// Mitsubishi GX Works2 project: msp_4   PLC: Q03UDV

PROGRAM MAIN
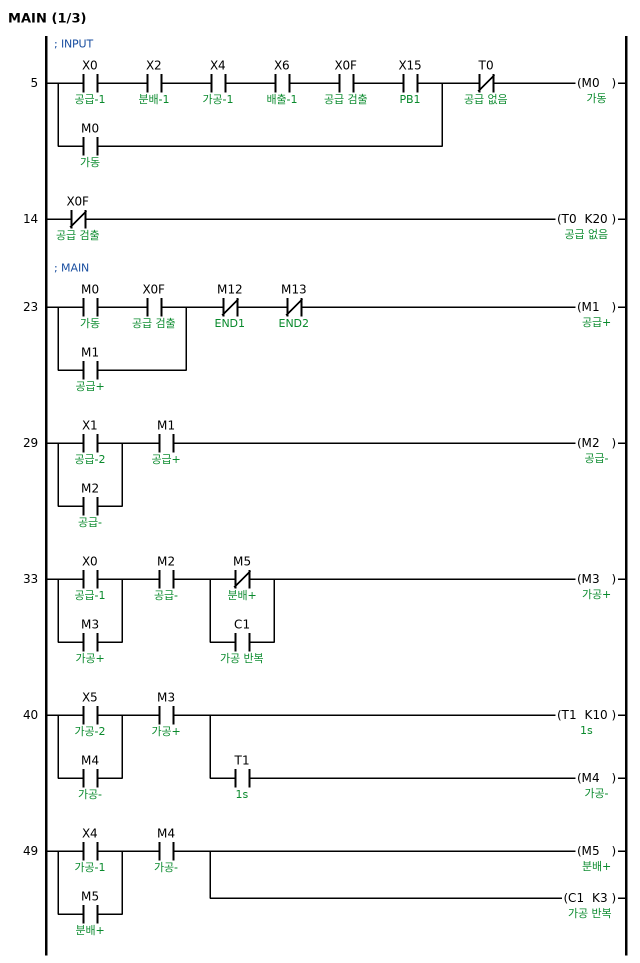
; INPUT
5     LD      X0  ; 공급-1
      AND     X2  ; 분배-1
      AND     X4  ; 가공-1
      AND     X6  ; 배출-1
      AND     X0F  ; 공급 검출
      AND     X15  ; PB1
      OR      M0  ; 가동
      ANI     T0  ; 공급 없음
      OUT     M0  ; 가동
14    LDI     X0F  ; 공급 검출
      OUT     T0 K20  ; 공급 없음
; MAIN
23    LD      M0  ; 가동
      AND     X0F  ; 공급 검출
      OR      M1  ; 공급+
      ANI     M12  ; END1
      ANI     M13  ; END2
      OUT     M1  ; 공급+
29    LD      X1  ; 공급-2
      OR      M2  ; 공급-
      AND     M1  ; 공급+
      OUT     M2  ; 공급-
33    LD      X0  ; 공급-1
      OR      M3  ; 가공+
      AND     M2  ; 공급-
      LDI     M5  ; 분배+
      OR      C1  ; 가공 반복
      ANB
      OUT     M3  ; 가공+
40    LD      X5  ; 가공-2
      OR      M4  ; 가공-
      AND     M3  ; 가공+
      OUT     T1 K10  ; 1s
      AND     T1  ; 1s
      OUT     M4  ; 가공-
49    LD      X4  ; 가공-1
      OR      M5  ; 분배+
      AND     M4  ; 가공-
      OUT     M5  ; 분배+
      OUT     C1 K3  ; 가공 반복
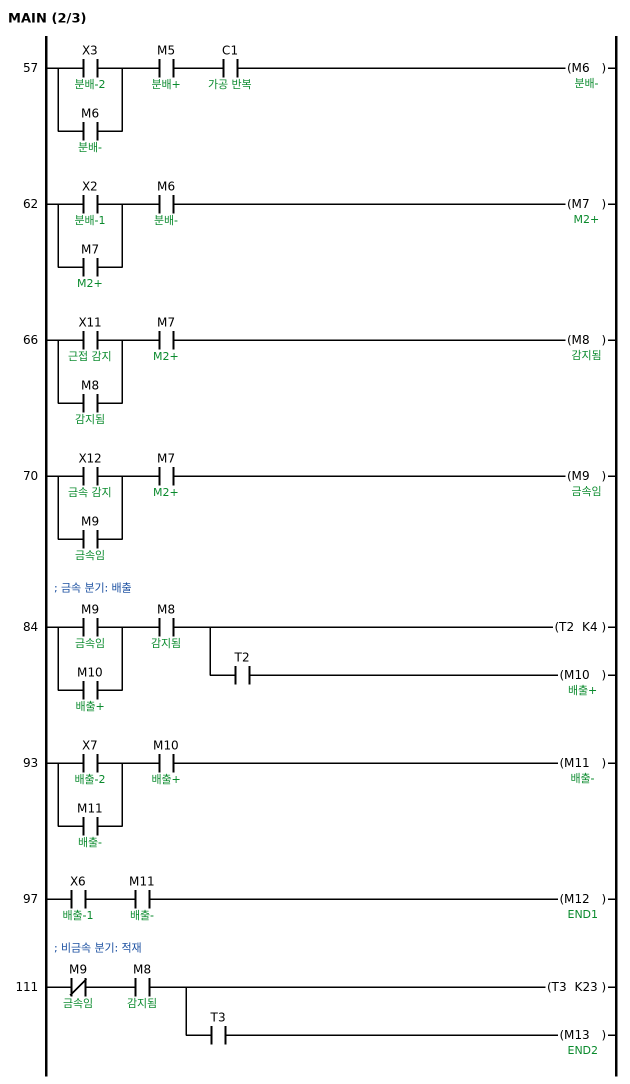
57    LD      X3  ; 분배-2
      OR      M6  ; 분배-
      AND     M5  ; 분배+
      AND     C1  ; 가공 반복
      OUT     M6  ; 분배-
62    LD      X2  ; 분배-1
      OR      M7  ; M2+
      AND     M6  ; 분배-
      OUT     M7  ; M2+
66    LD      X11  ; 근접 감지
      OR      M8  ; 감지됨
      AND     M7  ; M2+
      OUT     M8  ; 감지됨
70    LD      X12  ; 금속 감지
      OR      M9  ; 금속임
      AND     M7  ; M2+
      OUT     M9  ; 금속임
; 금속 분기: 배출
84    LD      M9  ; 금속임
      OR      M10  ; 배출+
      AND     M8  ; 감지됨
      OUT     T2 K4
      AND     T2
      OUT     M10  ; 배출+
93    LD      X7  ; 배출-2
      OR      M11  ; 배출-
      AND     M10  ; 배출+
      OUT     M11  ; 배출-
97    LD      X6  ; 배출-1
      AND     M11  ; 배출-
      OUT     M12  ; END1
; 비금속 분기: 적재
111   LDI     M9  ; 금속임
      AND     M8  ; 감지됨
      OUT     T3 K23
      AND     T3
      OUT     M13  ; END2
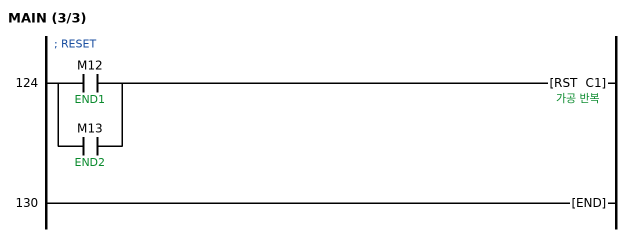
; RESET
124   LD      M12  ; END1
      OR      M13  ; END2
      RST     C1  ; 가공 반복
130   END
END_PROGRAM

PROGRAM OUTPUT
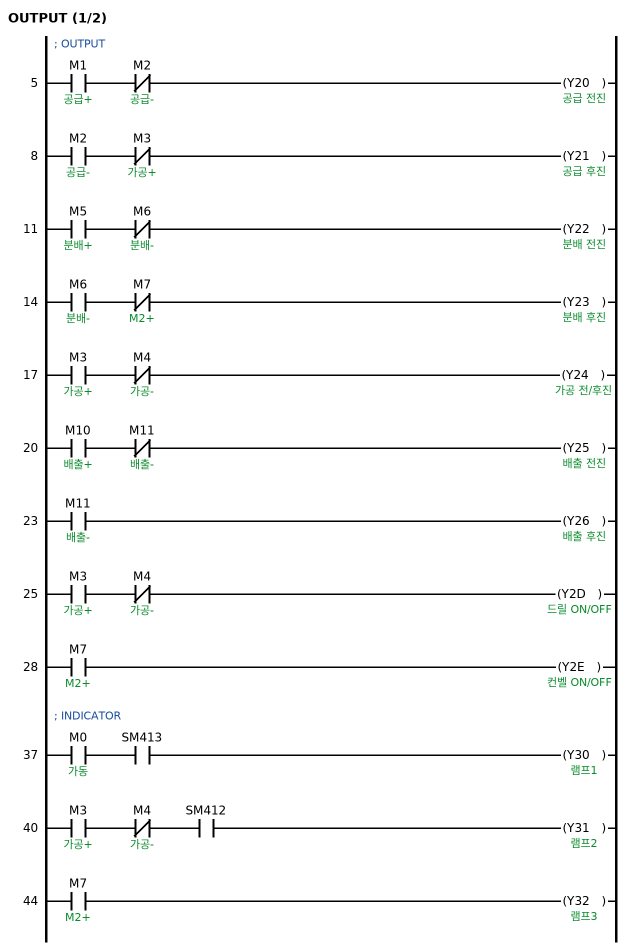
; OUTPUT
5     LD      M1  ; 공급+
      ANI     M2  ; 공급-
      OUT     Y20  ; 공급 전진
8     LD      M2  ; 공급-
      ANI     M3  ; 가공+
      OUT     Y21  ; 공급 후진
11    LD      M5  ; 분배+
      ANI     M6  ; 분배-
      OUT     Y22  ; 분배 전진
14    LD      M6  ; 분배-
      ANI     M7  ; M2+
      OUT     Y23  ; 분배 후진
17    LD      M3  ; 가공+
      ANI     M4  ; 가공-
      OUT     Y24  ; 가공 전/후진
20    LD      M10  ; 배출+
      ANI     M11  ; 배출-
      OUT     Y25  ; 배출 전진
23    LD      M11  ; 배출-
      OUT     Y26  ; 배출 후진
25    LD      M3  ; 가공+
      ANI     M4  ; 가공-
      OUT     Y2D  ; 드릴 ON/OFF
28    LD      M7  ; M2+
      OUT     Y2E  ; 컨벨 ON/OFF
; INDICATOR
37    LD      M0  ; 가동
      AND     SM413
      OUT     Y30  ; 램프1
40    LD      M3  ; 가공+
      ANI     M4  ; 가공-
      AND     SM412
      OUT     Y31  ; 램프2
44    LD      M7  ; M2+
      OUT     Y32  ; 램프3
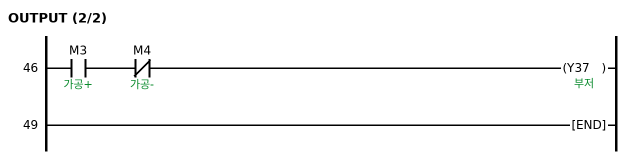
46    LD      M3  ; 가공+
      ANI     M4  ; 가공-
      OUT     Y37  ; 부저
49    END
END_PROGRAM

// device comments not shown above
X8  ; 스토퍼-1
X9  ; 스토퍼-2
X0A  ; 흡착-1
X0B  ; 흡착-2
X0C  ; 흡착 검출
X0D  ; 창고-1
X0E  ; 창고-2
X10  ; 공급 검출
X13  ; 스토퍼 감지
X14  ; 컨벨 인코더
X16  ; PB2
X17  ; PB3
X18  ; PB4
X19  ; PB5
X1A  ; PB6
X1B  ; PB7
X1C  ; PB8
X20  ; A 전진
X21  ; A 후진
X24  ; B 전진/후진
X2D  ; 가공 모터
Y27  ; 스토퍼 전/후진
Y28  ; 흡착 전진
Y29  ; 흡착 후진
Y2A  ; 흡착 ON/OFF
Y2B  ; 창고 전진
Y2C  ; 창고 후진
Y33  ; 램프4
Y34  ; 램프5
Y35  ; 램프6
Y36  ; 램프7
